METHOD PUBLIC updateCmds : BOOL
VAR_IN_OUT CONSTANT
	i_cartCtrlCmd : ST_SlaveArmCtrlCmds;
END_VAR
VAR
	i:INT;
END_VAR
m_cmdJntTrq:=i_cartCtrlCmd.m_cmdJntTrq;
m_cmdJntPos :=i_cartCtrlCmd.m_cmdJntPos;
m_cmdJntVel :=i_cartCtrlCmd.m_cmdJntVel;


// enable/disable joints
enable(i_cartCtrlCmd.m_jntEnableFlag);

// position/Velocity control
FOR i:=1 TO g_sJntNum DO 
	IF i_cartCtrlCmd.m_jntOPMode[i]=DriverOPMode_Pos THEN
		m_cmdJntTrq[i]:=0;
		m_cmdJntVel[i]:=0;
		m_cartJoints[i].updateCmd(DriverOPMode_Pos,m_cmdJntPos[i],m_cmdJntTrq[i],m_cmdJntVel[i]);
	ELSIF i_cartCtrlCmd.m_jntOPMode[i]=DriverOPMode_Vel THEN
		m_cmdJntTrq[i]:=0;
		m_cmdJntPos[i]:=0;
		m_cartJoints[i].updateCmd(DriverOPMode_Pos,m_cmdJntPos[i],m_cmdJntTrq[i],m_cmdJntVel[i]);
	ELSIF i_cartCtrlCmd.m_jntOPMode[i]=DriverOPMode_MZPos  THEN
		m_cmdJntTrq[i]:=0;
		m_cmdJntVel[i]:=0;
		//Input torque mode because the operating mode word for the contour position mode of the MingZhi driver is 1
		m_cartJoints[i].updateCmd(DriverOPMode_Trq,m_cmdJntPos[i],m_cmdJntTrq[i],m_cmdJntVel[i]);
	ELSIF i_cartCtrlCmd.m_jntOPMode[i]=DriverOPMode_cspMZ  THEN
		 m_cartJoints[i].updateCmd(DriverOPMode_cspMZ,m_cmdJntPos[i],m_cmdJntTrq[i],m_cmdJntVel[i]);
	ELSIF DriverOPMode_csvMZ = i_cartCtrlCmd.m_jntOPMode[i] THEN
		m_cartJoints[i].updateCmd(DriverOPMode_csvMZ,m_cmdJntPos[i],m_cmdJntTrq[i],m_cmdJntVel[i]);
	END_IF
END_FOR
END_METHOD

METHOD PUBLIC updateStatus : BOOL
VAR_INPUT
END_VAR
VAR
	i:INT;
END_VAR
// update joint data
FOR i:=1 TO g_sJntNum DO
	m_cartJoints[i].updateStatus();
END_FOR

//IO output   Horizontal laser IO output   Cross laser IO output
checkIO();


// get joint data
FOR i:=1 TO g_cartJntNum DO
	m_curMotorPos[i]:=m_cartJoints[i].motorPos;
	m_curLinkPos[i]:=m_cartJoints[i].linkPos;
	m_curLinkSingle[i]:=m_cartJoints[i].linkSingle;
	m_curJntPos[i]:=m_cartJoints[i].jntPos;
	m_curJntVel[i]:=m_cartJoints[i].jntVel;
	m_curJntTrq[i]:=m_cartJoints[i].jntTrq;
	m_rawJntCurrent[i]:=m_cartJoints[i].rawCurrent;
	m_filtJntCurrent[i]:=m_cartJoints[i].filtCurrent;
	m_cmdJntCurrent[i]:=m_cartJoints[i].cmdCurrent;
END_FOR
END_METHOD

END_FUNCTION_BLOCK

// ---- FBs_Robots/FB_CartJoint.TcPOU
FUNCTION_BLOCK FB_CartJoint EXTENDS FB_JointBase
VAR_INPUT
END_VAR
VAR_OUTPUT
END_VAR
VAR
	//Cart motor output IO
	m_cartMotorOutput AT %Q*	:ST_CartMotorOutput;
	
	m_cartMotorVelSongxia AT %I*  : DINT;

	m_cmdAcc:LREAL;
	
END_VAR

METHOD cmd2motorMZ : DINT
VAR_INPUT
	i_cmd:LREAL;
	i_controlCycleTime :LREAL;
END_VAR
cmd2motorMZ:=LREAL_TO_DINT(i_cmd / m_motorEnc2PosRatio);//*i_controlCycleTime
END_METHOD

METHOD PUBLIC enableMZ : BOOL
VAR_INPUT
END_VAR
IF (MZDriverStatusWord_SwitchOnDisable AND m_motorInputs.m_statusWord) = MZDriverStatusWord_SwitchOnDisable    THEN
	m_motorOutputs.m_controlWord:=DriverCtrlWord_INIT;
	enableMZ := FALSE;
ELSIF (MZDriverStatusWord_OperationEnbale AND m_motorInputs.m_statusWord) = MZDriverStatusWord_OperationEnbale THEN
	enableMZ :=  TRUE;
ELSIF (MZDriverStatusWord_SwitchOn AND m_motorInputs.m_statusWord) =  MZDriverStatusWord_SwitchOn THEN
	m_motorOutputs.m_controlWord:=DriverCtrlWord_OP;
	enableMZ :=  FALSE;
ELSIF (MZDriverStatusWord_ReadyToSwitchOn AND m_motorInputs.m_statusWord) = MZDriverStatusWord_ReadyToSwitchOn THEN
	m_motorOutputs.m_controlWord:=DriverCtrlWord_PREOP;
	enableMZ :=  FALSE;
ELSIF (MZDriverStatusWord_Fault AND m_motorInputs.m_statusWord) = MZDriverStatusWord_Fault THEN
	m_motorOutputs.m_controlWord:=DriverCtrlWord_FaultReset;
//ELSE
//	m_motorOutputs.m_controlWord:=DriverCtrlWord_INIT;
//	enable :=  FALSE;
END_IF
END_METHOD

METHOD PUBLIC init : BOOL
VAR_INPUT
	i_jntIdx :INT;
	i_controlCycleTime :LREAL;
END_VAR
m_jntIdx:=i_jntIdx;
m_cycleTime := i_controlCycleTime;

// hardware parameters
m_motorEncoderRes :=GVL_CartMotorParameters.g_incEncoderRes[i_jntIdx];
m_linkEncoderRes :=GVL_CartMotorParameters.g_absEncoderRes[i_jntIdx];
m_motorReduction :=GVL_CartMotorParameters.g_motorReduction[i_jntIdx];
m_linkEncoderReduction :=GVL_CartMotorParameters.g_absEncoderReduction[i_jntIdx];
m_trqConst :=GVL_CartMotorParameters.g_motorTrqConst[i_jntIdx];
m_maxCurrent :=GVL_CartMotorParameters.g_motorMaxCurrent[i_jntIdx];
m_motorDir :=GVL_CartMotorParameters.g_motorDir[i_jntIdx];								
m_minJntPos	:=GVL_CartMotorParameters.g_minJntPos[i_jntIdx];
m_maxJntPos	:=GVL_CartMotorParameters.g_maxJntPos[i_jntIdx];

//link encoder calibartion data
m_linkEncoderDir :=GVL_CartJointEncoderCaliData.g_asbEncoderDir[i_jntIdx];
m_minLinkEncoder :=GVL_CartJointEncoderCaliData.g_minLinkEncoder[ i_jntIdx] - m_linkEncoderDir*GVL_CartJointEncoderCaliData.g_linkEncLimitBuffer; // expand limit
m_maxLinkEncoder :=GVL_CartJointEncoderCaliData.g_maxLinkEncoder[ i_jntIdx] + m_linkEncoderDir*GVL_CartJointEncoderCaliData.g_linkEncLimitBuffer; // expand limit
m_caliLinkEncoder :=GVL_CartJointEncoderCaliData.g_caliLinkEncoder[ i_jntIdx];
m_linkEncCaliJntPos :=GVL_CartJointEncoderCaliData.g_linkEncCaliJntPos[i_jntIdx];
m_linkEncZeroCross :=GVL_CartJointEncoderCaliData.g_linkEncZeroCross[ i_jntIdx];
m_multiCycles :=GVL_CartJointEncoderCaliData.g_multipleCyclesJoint[i_jntIdx];

// convert cali link encoder if joint cross zero
IF 1=m_linkEncZeroCross THEN
	IF 1=m_linkEncoderDir AND m_caliLinkEncoder < m_minLinkEncoder THEN
		m_caliLinkEncoder := GVL_CartJointEncoderCaliData.g_caliLinkEncoder[ i_jntIdx] + m_linkEncoderRes;
	ELSIF -1=m_linkEncoderDir AND m_caliLinkEncoder < m_maxLinkEncoder THEN
		m_caliLinkEncoder := GVL_CartJointEncoderCaliData.g_caliLinkEncoder[ i_jntIdx] + m_linkEncoderRes;
	END_IF
END_IF

// macro data
m_trq2CurrentRatio:=m_motorDir * 1000.0/(m_trqConst*m_motorReduction);
m_current2TrqRatio:=m_motorDir * (m_trqConst*m_motorReduction)/1000.0;
m_linkEnc2PosRatio := 2*PI*m_linkEncoderDir/(m_linkEncoderReduction*m_linkEncoderRes);
m_motorEnc2PosRatio := 2*PI * m_motorDir/(m_motorReduction * m_motorEncoderRes);


// motor data init
m_rawJntVel :=0;
m_curJntVel:=0;
m_curJntTrq :=0;
m_rawCurrent :=0;
m_filtCurrent :=0;
m_cmdJntVel :=0.0;
m_cmdJntTrq :=0.0;
m_cmdCurrent := 0.0;

// filter init
m_jntVelLpf.init(1, GVL_CartControlParameters.g_curJntVelLpfCutoffFreq, g_cartCtrlFreq);
m_cmdTrqLpf.init(1, GVL_CartControlParameters.g_cmdJntTrqLpfCutoffFreq, g_cartCtrlFreq);
m_curTrqLpf.init(1, GVL_CartControlParameters.g_curJntTrqLpfCutoffFreq, g_cartCtrlFreq);

// driver init value
m_motorOutputs.m_controlWord:=DriverCtrlWord_INIT;
m_motorOutputs.m_opMode:=INT_TO_SINT(DriverOPMode_Pos);
m_motorOutputs.m_cmdCurrent:=0;
m_motorOutputs.m_cmdMotorEncoder:=m_motorInputs.m_motorEncoder;
END_METHOD

METHOD PUBLIC updateCmd : BOOL
VAR_INPUT
	i_opMode : E_DriverOPMode;
	i_cmdPos :LREAL;
	i_cmdTrq :LREAL;
	i_cmdVel :LREAL;
END_VAR
VAR
	i:INT;
END_VAR
m_motorOutputs.m_opMode:=INT_TO_SINT( i_opMode);

// pos mode
IF i_opMode = DriverOPMode_Pos OR i_opMode = DriverOPMode_cspMZ  THEN
	m_motorOutputs.m_cmdCurrent:=0;
	m_cmdJntPos :=i_cmdPos;
	m_cartMotorOutput.m_cmdVelMzVelMode :=0;
	m_motorOutputs.m_cmdMotorEncoder :=motorPos2Enc(m_cmdJntPos);
ELSIF i_opMode = DriverOPMode_Vel THEN
	m_cmdJntVel := i_cmdVel;
	m_cartMotorOutput.m_cmdVelMzVelMode := cmd2motorMZ(m_cmdJntVel, g_cartCtrlCycleTime);
	
ELSIF i_opMode = DriverOPMode_Trq THEN   //Here the torque mode is equal to the contour position mode of the MingZhi driver
	m_cmdJntVel := i_cmdVel;
	m_cmdAcc:=i_cmdVel*2;
	m_cmdJntPos:=i_cmdPos;
	m_cartMotorOutput.m_cmdAccMz :=cmd2motorMZ(m_cmdAcc, g_cartCtrlCycleTime);
	//m_cartMotorOutput.m_cmdVelMz := cmd2motorMZ(m_cmdJntVel, g_cartCtrlCycleTime);
	m_motorOutputs.m_cmdMotorEncoder := motorPos2Enc(m_cmdJntVel);
ELSIF i_opMode = DriverOPMode_csvMZ THEN
	m_cmdJntVel := i_cmdVel;
	m_cartMotorOutput.m_cmdVelMzVelMode := cmd2motorMZ(m_cmdJntVel, g_cartCtrlCycleTime);
	m_cartMotorOutput.m_cmdVelMax := 419430400;
END_IF
END_METHOD

METHOD PUBLIC updateStatus : BOOL
VAR_INPUT
END_VAR
// compute joint position
m_curLinkPos:= linkEnc2Pos();
m_curMotorPos:=motorEnc2Pos();
m_curLinkSingle := m_curLinkPos - 2*PI* m_linkEncCycles;

// Cart joint1-4 have no link enconder, use motor position
IF m_jntIdx <= 8 THEN
	m_curJntPos := m_curMotorPos;
ELSE
	m_curJntPos := m_curLinkPos;
END_IF

// compute joint velocity
m_curVelCalCycles := m_curVelCalCycles+1;
IF m_curVelCalCycles > m_velCalcCycles THEN
	m_rawJntVel:= (m_curJntPos-m_lastJntPos)/(m_cycleTime*m_velCalcCycles);
	m_curJntVel := m_jntVelLpf.run(m_rawJntVel);
	m_lastJntPos :=m_curJntPos;	
	m_curVelCalCycles:=1;
END_IF

IF m_jntIdx = 3 OR  m_jntIdx = 4 THEN
	m_curJntVel := m_cartMotorVelSongxia * m_motorEnc2PosRatio;
END_IF

// current and torque
m_rawCurrent := m_motorInputs.m_current;
m_filtCurrent := m_curTrqLpf.run(m_rawCurrent);
m_curJntTrq := m_filtCurrent * m_current2TrqRatio;
END_METHOD

END_FUNCTION_BLOCK

// ---- FBs_Robots/FB_JointBase.TcPOU
FUNCTION_BLOCK FB_JointBase
VAR_INPUT
END_VAR
VAR_OUTPUT
END_VAR
VAR
	// arm and joint index
	m_armIdx :INT;
	m_jntIdx :INT;
	
	// motor IO
	m_motorInputs AT%I*	:ST_MotorInputs;
	m_motorOutputs AT%Q* :ST_MotorOutputs;
	
	// cycle time
	m_cycleTime :LREAL;
	
	// calibrated link encoder data
	m_minLinkEncoder :DINT;
	m_maxLinkEncoder :DINT;
	m_caliLinkEncoder :DINT;
	m_linkEncCaliJntPos :LREAL;
	m_linkEncZeroCross :INT;
	m_initMotorEnc : DINT;
	m_multiCycles :INT;
	
	// joint position from link encoder after power on
	m_initLinkPos :LREAL;
	
	// data for link encoder multiple cycles
	m_lastLinkEncoder :DINT;
	m_linkEncCycles:INT;
	
	// device paramters
	m_motorEncoderRes :DINT;
	m_linkEncoderRes :DINT;
	m_linkEncLimitBuffer : DINT;
	m_motorReduction :LREAL;
	m_linkEncoderReduction :LREAL;
	m_trqConst :LREAL;
	m_maxCurrent :LREAL;
	m_motorDir :INT;								
	m_linkEncoderDir :INT;
	m_minJntPos: LREAL;
	m_maxJntPos: LREAL;
	
	// macro defined data for quick calculation
	m_trq2CurrentRatio:LREAL;
	m_current2TrqRatio:LREAL;
	m_linkEnc2PosRatio :LREAL;
	m_motorEnc2PosRatio :LREAL;
	
	// joint data
	m_curMotorPos :LREAL;
	m_curLinkPos :LREAL;
	m_curLinkSingle :LREAL;//[0-360]
	m_curJntPos	:LREAL;
	m_curJntVel :LREAL;
	m_rawJntVel :LREAL;
	m_curJntTrq :	LREAL;
	m_rawCurrent : LREAL;
	m_filtCurrent : LREAL;
	m_cmdJntPos :LREAL;
	m_cmdJntVel :LREAL;
	m_cmdJntTrq :LREAL;
	m_cmdCurrent : LREAL;
	m_lastJntPos :LREAL;
	
	// velocity filter
	m_jntVelLpf :FB_LowPassFilter;
	
	// command torque filter
	m_curTrqLpf : FB_LowPassFilter;
	m_cmdTrqLpf :FB_LowPassFilter;
	
	// velocity is calculated every (m_velCalcCycles) control cycles
	// TODO: insturment joint motor can not reach 4k now, so calculate their velocity with 1k frequency, need to remove later
	m_velCalcCycles :INT :=1;
	m_curVelCalCycles :INT :=1;
	
	// SDO writer
	m_opModeSDOWrite:FB_EcCoESdoWrite;
	m_MotorCurrentSDOWrite:FB_EcCoESdoWrite;
	
END_VAR

PROPERTY cmdCurrent : LREAL
GET
cmdCurrent:=m_cmdCurrent;
END_GET
END_PROPERTY

METHOD PUBLIC disable : BOOL
VAR_INPUT
END_VAR
m_motorOutputs.m_controlWord:=DriverCtrlWord_INIT;
disable:=true;
END_METHOD

METHOD PUBLIC enable : BOOL
VAR_INPUT
END_VAR
IF DriverStatusWord_INIT = m_motorInputs.m_statusWord THEN
	m_motorOutputs.m_controlWord:=DriverCtrlWord_PREOP;
	enable := FALSE;
ELSIF DriverStatusWord_PREOP = m_motorInputs.m_statusWord THEN
	m_motorOutputs.m_controlWord:=DriverCtrlWord_OP;
	enable :=  FALSE;
ELSIF DriverStatusWord_OP = m_motorInputs.m_statusWord THEN
	enable :=  TRUE;
//ELSE
//	m_motorOutputs.m_controlWord:=DriverCtrlWord_INIT;
//	enable :=  FALSE;
END_IF
END_METHOD

PROPERTY filtCurrent : LREAL
GET
filtCurrent:=m_filtCurrent;
END_GET
END_PROPERTY

METHOD PUBLIC initJntPos : BOOL
VAR_INPUT
END_VAR
m_lastLinkEncoder :=m_motorInputs.m_linkEncoder;
m_linkEncCycles:=0;
m_curLinkPos :=linkEnc2Pos();
m_initLinkPos:=m_curLinkPos;
m_initMotorEnc :=m_motorInputs.m_motorEncoder;
m_curMotorPos:=motorEnc2Pos();
m_curJntPos := m_curMotorPos;
m_cmdJntPos :=m_curJntPos;	
m_lastJntPos :=m_curJntPos;
END_METHOD

PROPERTY initLinkPos : lreal
GET
initLinkPos:=m_initLinkPos;
END_GET
SET
m_initLinkPos:=initLinkPos;
END_SET
END_PROPERTY

METHOD PUBLIC isEnabled : BOOL
VAR_INPUT
END_VAR
isEnabled :=(DriverStatusWord_OP = m_motorInputs.m_statusWord);
END_METHOD

PROPERTY jntPos : LREAL
GET
jntPos := m_curJntPos;
END_GET
END_PROPERTY

PROPERTY jntTrq : LREAL
GET
jntTrq:=m_curJntTrq;
END_GET
END_PROPERTY

PROPERTY jntVel : LREAL
GET
jntVel := m_curJntVel;
END_GET
END_PROPERTY

METHOD PROTECTED linkEnc2Pos : LREAL
VAR_INPUT
END_VAR
VAR
	incLinkPos :LREAL;
	newLinkEnc :DINT;
END_VAR
// cycle check
IF 1=m_multiCycles THEN
	IF (m_motorInputs.m_linkEncoder - m_lastLinkEncoder)*m_linkEncoderDir < -m_linkEncoderRes/2 THEN
		m_linkEncCycles :=m_linkEncCycles+1;
	ELSIF (m_motorInputs.m_linkEncoder - m_lastLinkEncoder)*m_linkEncoderDir > m_linkEncoderRes/2 THEN
		m_linkEncCycles :=m_linkEncCycles-1;
	END_IF
END_IF
m_lastLinkEncoder:=m_motorInputs.m_linkEncoder;

// convert link encoder if joint cross zero
newLinkEnc := m_motorInputs.m_linkEncoder;
IF 1=m_linkEncZeroCross AND 0 = m_multiCycles THEN
	IF 1=m_linkEncoderDir AND m_motorInputs.m_linkEncoder < m_minLinkEncoder THEN
		newLinkEnc := m_motorInputs.m_linkEncoder + m_linkEncoderRes;
	ELSIF -1=m_linkEncoderDir AND m_motorInputs.m_linkEncoder < m_maxLinkEncoder THEN
		newLinkEnc := m_motorInputs.m_linkEncoder + m_linkEncoderRes;
	END_IF
END_IF

// motion from calibrated points
incLinkPos := (newLinkEnc-m_caliLinkEncoder)*m_linkEnc2PosRatio;

// absolute joint position
linkEnc2Pos := incLinkPos + m_linkEncCaliJntPos + 2*PI* m_linkEncCycles;
END_METHOD

PROPERTY PUBLIC linkPos : LREAL
GET
linkPos:=m_curLinkPos;
END_GET
END_PROPERTY

PROPERTY linkSingle : LREAL
GET
linkSingle :=m_curLinkSingle;
END_GET
END_PROPERTY

METHOD PROTECTED motorEnc2Pos : LREAL
VAR_INPUT
END_VAR
motorEnc2Pos:= (m_motorInputs.m_motorEncoder-m_initMotorEnc)* m_motorEnc2PosRatio +m_initLinkPos;
END_METHOD

PROPERTY PUBLIC motorPos : LREAL
GET
motorPos := m_curMotorPos;
END_GET
END_PROPERTY

METHOD PROTECTED motorPos2Enc : DINT
VAR_INPUT
	i_jntPos :LREAL;
END_VAR

VAR
END_VAR

motorPos2Enc := LREAL_TO_DINT((i_jntPos-m_initLinkPos)/m_motorEnc2PosRatio + m_initMotorEnc);
END_METHOD

PROPERTY rawCurrent : LREAL
GET
rawCurrent := m_rawCurrent;
END_GET
END_PROPERTY

METHOD PROTECTED singleCyclePos : LREal
VAR_INPUT
END_VAR
VAR
	cycles :lreal;
END_VAR
cycles := ABS(FLOOR( m_curJntPos/g_2pi));
IF m_curJntPos<0 THEN
	singleCyclePos := m_curJntPos+cycles*g_2pi;
ELSE
	singleCyclePos := m_curJntPos-cycles*g_2pi;
END_IF
END_METHOD

METHOD PUBLIC updateCmds : BOOL
VAR_INPUT
	i_opMode : E_DriverOPMode;
	i_cmdPos :LREAL;
	i_cmdTrq :LREAL;
END_VAR
VAR
	filtCmdTrq :LREAL;
END_VAR
m_motorOutputs.m_opMode:=INT_TO_SINT( i_opMode);
// pos mode
IF i_opMode = DriverOPMode_Pos THEN
	m_motorOutputs.m_cmdCurrent:=0;
	m_cmdTrqLpf.reset();	
//	i_cmdPos:=LIMIT(m_minJntPos, i_cmdPos, m_maxJntPos); // May cause position jump, Do this in safety check. 
	m_cmdJntPos :=i_cmdPos;
	m_motorOutputs.m_cmdMotorEncoder :=motorPos2Enc(m_cmdJntPos);
ELSIF i_opMode = DriverOPMode_Trq THEN
	filtCmdTrq:=m_cmdTrqLpf.run(i_cmdTrq);
	m_motorOutputs.m_cmdCurrent:=LREAL_TO_DINT(LIMIT(-m_maxCurrent, filtCmdTrq*m_trq2CurrentRatio,m_maxCurrent));
	m_motorOutputs.m_cmdMotorEncoder :=m_motorInputs.m_motorEncoder; 
END_IF
m_cmdCurrent:=m_motorOutputs.m_cmdCurrent;
END_METHOD

METHOD PUBLIC updateStatus : BOOL
VAR_INPUT
END_VAR
// compute joint position
m_curLinkPos:= linkEnc2Pos();
m_curMotorPos:=motorEnc2Pos();
m_curJntPos := m_curMotorPos;
m_curLinkSingle := singleCyclePos();

// compute joint velocity
m_curVelCalCycles := m_curVelCalCycles+1;
IF m_curVelCalCycles > m_velCalcCycles THEN
	m_rawJntVel:= (m_curJntPos-m_lastJntPos)/(m_cycleTime*m_velCalcCycles);
	m_curJntVel := m_jntVelLpf.run(m_rawJntVel);
	m_lastJntPos :=m_curJntPos;	
	m_curVelCalCycles:=1;
END_IF


// current and torque
m_rawCurrent := m_motorInputs.m_current;
m_filtCurrent := m_curTrqLpf.run(m_rawCurrent);
m_curJntTrq := m_filtCurrent * m_current2TrqRatio;
END_METHOD

END_FUNCTION_BLOCK

// ---- FBs_CartControlles/FB_CartCtrlAdjust.TcPOU
FUNCTION_BLOCK FB_CartCtrlAdjust EXTENDS FB_CartCtrlBase
VAR_INPUT
END_VAR
VAR_OUTPUT
END_VAR
VAR

	m_joystickSignal: Vec8d;	
	m_fiducialValue:INT:= 512;
	m_joystickRange:INT:=430;
	m_joystickDir: Vec8i:=[1,1,1,1,-1,-1,1,1];
	m_joystickVelInc: Vec8d;
	m_actJntPos: Vec8d;
	m_tarPosInc: Vec8d;
	m_lastPosInc: Vec8d;
	m_tarCartPos: Vec8d;
	m_trajJntPos : Vec8d;
	m_tarJntPos : Vec8d;
	m_initActJntPos: Vec8d;
	m_initActCartPos: Vec8d;
	m_veiwAngle : LREAL;
	m_jntPosReachLimit : Vec8b;
	m_maxJntPos : vec8d;

	m_carJntSoftwareLimit :ARRAY [5..8] OF LREAL := [0.005, 2*g_deg2Rad, 0.005, 2*g_deg2Rad];
	
	// time threshold to 5-8joint after it's enabled
	m_cartAdjustStartWaitTime :LREAL := 0.3;
	
	//adjust start  time 
	m_adjustStartTime :LREAL;
	
	// filter cut-off frequency for cart drive force 
	m_cmdJoystickLpfCutoffFreq : LREAL :=8;
	m_cartCtrlFreq :LREAL:=8000;
	
	m_Vel : LREAL;
	m_velDir : INT;
	m_jntOTG :ARRAY[1..8] OF FB_secOrdTrajFilter;
END_VAR

// override this function in each exact controller
METHOD PROTECTED calcCmdJntPos : BOOL
VAR_IN_OUT CONSTANT
	// slave cart joint data
	i_slaveCart :FB_SlaveCart;
END_VAR

VAR
	i:INT;
END_VAR
//In this method, 5 represents the pillar postion , 6 represents the beam rotation angle ,7 represents the beam stretch position ,8 represents the overhang angle
m_adjustStartTime :=LIMIT(0, m_adjustStartTime + g_cartCtrlCycleTime, 1);
m_actJntPos := i_slaveCart.curJntPos;
m_actJntPos[7] := i_slaveCart.curJntPos[7] + GVL_CartControlParameters.g_curBeamStretchJntInitPos;
m_veiwAngle := m_actJntPos[6] + m_actJntPos[8];

IF m_adjustStartTime > m_cartAdjustStartWaitTime THEN
	FOR i:= 1 TO 4 BY 1 DO
		m_joystickSignal[i] := i_slaveCart.m_joystickSignal[i] - m_fiducialValue;
		m_joystickVelInc[i+4] := m_joystickSignal[i]/m_joystickRange*m_joystickDir[i+4]*GVL_CartControlParameters.g_maxCartVel[i];
		m_tarPosInc[i+4] := m_tarPosInc[i+4] + m_joystickVelInc[i+4] * g_cartCtrlCycleTime;
	END_FOR
	
	m_tarCartPos[5] := m_initActJntPos[5] + m_tarPosInc[5];
	IF i_slaveCart.m_ctrlEnable.m_cameraJoystickEnable THEN
		m_tarCartPos[6] := m_initActCartPos[6] + m_tarPosInc[6]*COS(m_veiwAngle)+m_tarPosInc[7]*SIN(m_veiwAngle);
		m_tarCartPos[7] := m_initActCartPos[7] - m_tarPosInc[6]*SIN(m_veiwAngle)+m_tarPosInc[7]*COS(m_veiwAngle);
	ELSE
		m_tarCartPos[6] := m_initActCartPos[6] + m_tarPosInc[6];
		m_tarCartPos[7] := m_initActCartPos[7] + m_tarPosInc[7];
	END_IF
	m_tarCartPos[8] := m_initActJntPos[8] + m_tarPosInc[8];
	
	IF i_slaveCart.m_ctrlEnable.m_heightLimitAdjustEnable THEN
		m_trajJntPos[5] := m_tarCartPos[5];
	ELSE
		m_trajJntPos[5] := LIMIT(GVL_CartMotorParameters.g_minJntPos[5], m_tarCartPos[5], MAX(m_actJntPos[5],i_slaveCart.m_cartDataFromUI.m_standColumnHightLimit));
	END_IF
	m_trajJntPos[6] := atan2( m_tarCartPos[6], m_tarCartPos[7]);
	m_trajJntPos[7] := m_tarCartPos[7]/COS(m_trajJntPos[6]) - GVL_CartControlParameters.g_curBeamStretchJntInitPos;
	m_trajJntPos[8] := m_tarCartPos[8] -  (m_trajJntPos[6] - m_initActJntPos[6]);
	m_jntPosReachLimit := calcCmdReachLimit();
	m_jntEnableFlag := faultDetect(i_slaveCart.curJntPos);
	FOR i := 5 TO 8 DO 
		m_tarJntPos[i] := LIMIT(GVL_CartMotorParameters.g_minJntPos[i] + m_carJntSoftwareLimit[i], m_trajJntPos[i], GVL_CartMotorParameters.g_maxJntPos[i] - m_carJntSoftwareLimit[i]) ;
		m_jntOTG[i].run(i_targetPos:= m_trajJntPos[i], i_targetVel:= 0.0, o_cmdAcc=> , o_cmdVel=> , o_cmdPos=>m_cmdJntPos[i] );
	END_FOR
END_IF
END_METHOD

METHOD calcCmdReachLimit : vec8b
VAR_INPUT
END_VAR

VAR
	i : INT;
END_VAR

FOR i := 5 TO g_cartJntNum DO
	IF (GVL_CartMotorParameters.g_minJntPos[i] + m_carJntSoftwareLimit[i]) >= m_trajJntPos[i] THEN
		IF (m_tarPosInc[i] - m_lastPosInc[i]) <0 THEN
			m_tarPosInc[i] := m_lastPosInc[i];
		END_IF
		calcCmdReachLimit[i] := TRUE;
	
	ELSIF m_trajJntPos[i]>=(m_maxJntPos[i] - m_carJntSoftwareLimit[i]) THEN
		IF (m_tarPosInc[i] - m_lastPosInc[i]) >0 THEN
			m_tarPosInc[i] := m_lastPosInc[i];
		END_IF
		calcCmdReachLimit[i] := TRUE;
	END_IF
	m_lastPosInc[i] := m_tarPosInc[i];
END_FOR
END_METHOD

METHOD faultDetect : vec8i
VAR_INPUT
	curJntPos : vec8d;
END_VAR
faultDetect[5] := BOOL_TO_INT( NOT SafetyCheck.m_safetyCheckData.m_cartStandColumnErr);
faultDetect[6] := BOOL_TO_INT( NOT SafetyCheck.m_safetyCheckData.m_cartAdjustErr);
faultDetect[7] := BOOL_TO_INT( NOT SafetyCheck.m_safetyCheckData.m_cartAdjustErr);
faultDetect[8] := BOOL_TO_INT( NOT SafetyCheck.m_safetyCheckData.m_cartAdjustErr);

IF SafetyCheck.m_safetyCheckData.m_cartStandColumnErr THEN
	m_trajJntPos[5] :=curJntPos[5];
END_IF
IF SafetyCheck.m_safetyCheckData.m_cartAdjustErr THEN
	m_trajJntPos[6] :=curJntPos[6];
	m_trajJntPos[7] :=curJntPos[7];
	m_trajJntPos[8] :=curJntPos[8];
END_IF
END_METHOD

// override this function in each exact controller
// NOTICE: set joint control mode here, and do some initialization if needed
METHOD PUBLIC init : BOOL
VAR_IN_OUT CONSTANT
	i_slaveCart	:FB_SlaveCart;
END_VAR
VAR_IN_OUT 
	r_cartCtrlCmd :ST_SlaveArmCtrlCmds;
END_VAR
VAR
	i:INT;
END_VAR
// check if to hold the command joint position unchanged
//m_holdLastCmds := checkToHoldLastCmds(i_slaveCart);
m_holdLastCmds := checkToHoldLastCmds(i_slaveCart);
SUPER^.init(i_slaveCart,r_cartCtrlCmd);

m_jntEnableFlag[5] := BOOL_TO_INT( NOT SafetyCheck.m_safetyCheckData.m_cartStandColumnErr);
m_jntEnableFlag[6] := BOOL_TO_INT( NOT SafetyCheck.m_safetyCheckData.m_cartAdjustErr);
m_jntEnableFlag[7] := BOOL_TO_INT( NOT SafetyCheck.m_safetyCheckData.m_cartAdjustErr);
m_jntEnableFlag[8] := BOOL_TO_INT( NOT SafetyCheck.m_safetyCheckData.m_cartAdjustErr);

m_jntOPMode[5]:= DriverOPMode_cspMZ;
m_jntOPMode[6]:= DriverOPMode_Pos;
m_jntOPMode[7]:= DriverOPMode_Pos;
m_jntOPMode[8]:= DriverOPMode_Pos;

m_joystickSignal := g_zeroVec8d;
m_tarPosInc := g_zeroVec8d;
m_trajJntPos := g_zeroVec8d;
m_lastPosInc := g_zeroVec8d;
m_jntPosReachLimit := g_zeroVec8b;

m_maxJntPos := GVL_CartMotorParameters.g_maxJntPos;
m_maxJntPos[5] := i_slaveCart.m_cartDataFromUI.m_standColumnHightLimit;

m_initActJntPos:=m_cmdJntPos;//i_slaveCart.curJntPos;
m_initActCartPos[6] := (m_initActJntPos[7] + GVL_CartControlParameters.g_curBeamStretchJntInitPos) * SIN(m_initActJntPos[6]);
m_initActCartPos[7] := (m_initActJntPos[7] + GVL_CartControlParameters.g_curBeamStretchJntInitPos) * COS(m_initActJntPos[6]);

FOR i := 1 TO 4 BY 1 DO
	m_jntOTG[i+4].init(i_curCmdPos:= m_cmdJntPos[i+4], i_curCmdVel:= 0, i_maxV:=GVL_CartControlParameters.g_maxJntVel[i+4] , i_maxA:=GVL_CartControlParameters.g_maxJntAcc[i+4] , i_Ts:=g_cartCtrlCycleTime );
END_FOR

m_adjustStartTime := 0;
// update commands to arm
copyCmds(r_cartCtrlCmd);
END_METHOD

PROPERTY jntPosReachLimit : vec8b
GET
jntPosReachLimit := m_jntPosReachLimit;
END_GET
END_PROPERTY

END_FUNCTION_BLOCK

// ---- FBs_CartControlles/FB_CartCtrlSlowDown.TcPOU
FUNCTION_BLOCK FB_CartCtrlSlowDown EXTENDS FB_CartCtrlBase
VAR_INPUT
END_VAR
VAR_OUTPUT
END_VAR
VAR

	m_tarPosInc: Vec8d;
	m_trajVel : Vec8d;
	m_initVel : Vec8d;
	m_initPos : Vec8d;
	m_initDec : Vec8d;
	
	//slow down and stop time
	m_incSlowStopTime :LREAL;
	m_slowStopTime :LREAL :=0.5;
	
	// filter cut-off frequency for cart drive force 
	m_cmdJoystickLpfCutoffFreq : LREAL :=8;
	m_cartCtrlFreq :LREAL:=8000;
END_VAR

// override this function in each exact controller
METHOD PROTECTED calcCmdJntPos : BOOL
VAR_IN_OUT CONSTANT
	// slave cart joint data
	i_slaveCart :FB_SlaveCart;
END_VAR

VAR
	i:INT;
END_VAR
//In this method, 5 represents the pillar postion , 6 represents the beam rotation angle ,7 represents the beam stretch position ,8 represents the overhang angle
m_incSlowStopTime :=LIMIT(0, m_incSlowStopTime + g_cartCtrlCycleTime, 1);

FOR i := 5 TO 8 BY 1 DO
	m_trajVel[i] := m_initVel[i] - m_initDec[i] * m_incSlowStopTime;
	IF sign(m_trajVel[i]) <> sign(m_initVel[i]) THEN
		m_trajVel[i]:=0;
	END_IF
	m_tarPosInc[i] := m_tarPosInc[i] + m_trajVel[i] * g_cartCtrlCycleTime;
	m_cmdJntPos[i] := m_initPos[i] + m_tarPosInc[i];
END_FOR

IF m_incSlowStopTime >= m_slowStopTime THEN//m_slowStopTime THEN
	m_isFinished := TRUE;
END_IF
END_METHOD

// override this function in each exact controller
METHOD PROTECTED calcCmdJntVel : BOOL
VAR_IN_OUT CONSTANT
	// slave cart joint data
	i_slaveCart :FB_SlaveCart;
END_VAR

VAR
	i:INT;
END_VAR
//In this method, 5 represents the pillar postion , 6 represents the beam rotation angle ,7 represents the beam stretch position ,8 represents the overhang angle
m_incSlowStopTime :=LIMIT(0, m_incSlowStopTime + g_cartCtrlCycleTime, 1);

FOR i := 3 TO 4 BY 1 DO
	m_trajVel[i] := m_initVel[i] - m_initDec[i] * m_incSlowStopTime;
	IF sign(m_trajVel[i]) <> sign(m_initVel[i]) THEN
		m_trajVel[i]:=0;
	END_IF
	m_cmdJntVel[i] := LIMIT(-GVL_CartControlParameters.g_maxJntVel[i], m_trajVel[i]  , GVL_CartControlParameters.g_maxJntVel[i]);
END_FOR

IF m_incSlowStopTime >= m_slowStopTime THEN//m_slowStopTime THEN
	m_isFinished := TRUE;
END_IF
END_METHOD

// override this function in each exact controller
// NOTICE: set joint control mode here, and do some initialization if needed
METHOD PUBLIC init : BOOL
VAR_IN_OUT CONSTANT
	i_slaveCart	:FB_SlaveCart;
END_VAR
VAR_IN_OUT 
	r_cartCtrlCmd :ST_SlaveArmCtrlCmds;
END_VAR
m_cmdJntPos:=r_cartCtrlCmd.m_cmdJntPos;
m_initPos := m_cmdJntPos;

m_jntEnableFlag :=r_cartCtrlCmd.m_jntEnableFlag;

m_jntOPMode[3]:= DriverOPMode_csvMZ;
m_jntOPMode[4]:= DriverOPMode_csvMZ;
m_jntOPMode[5]:= DriverOPMode_cspMZ;
m_jntOPMode[6]:= DriverOPMode_Pos;
m_jntOPMode[7]:= DriverOPMode_Pos;
m_jntOPMode[8]:= DriverOPMode_Pos;

m_trajVel[3] := 0;
m_trajVel[4] := 0;
m_trajVel[5] := 0;
m_trajVel[6] := 0;
m_trajVel[7] := 0;
m_trajVel[8] := 0;

m_tarPosInc[3] := 0;
m_tarPosInc[4] := 0;
m_tarPosInc[5] := 0;
m_tarPosInc[6] := 0;
m_tarPosInc[7] := 0;
m_tarPosInc[8] := 0;


m_incSlowStopTime := 0;

m_initVel[3] := LIMIT(-GVL_CartControlParameters.g_maxJntVel[3], i_slaveCart.curJntVel[3], GVL_CartControlParameters.g_maxJntVel[3]);
m_initVel[4] := LIMIT(-GVL_CartControlParameters.g_maxJntVel[4], i_slaveCart.curJntVel[4], GVL_CartControlParameters.g_maxJntVel[4]);
m_initVel[5] := LIMIT(-GVL_CartControlParameters.g_maxJntVel[5], i_slaveCart.curJntVel[5], GVL_CartControlParameters.g_maxJntVel[5]);
m_initVel[6] := LIMIT(-GVL_CartControlParameters.g_maxJntVel[6], i_slaveCart.curJntVel[6], GVL_CartControlParameters.g_maxJntVel[6]);
m_initVel[7] := LIMIT(-GVL_CartControlParameters.g_maxJntVel[7], i_slaveCart.curJntVel[7], GVL_CartControlParameters.g_maxJntVel[7]);
m_initVel[8] := LIMIT(-GVL_CartControlParameters.g_maxJntVel[8], i_slaveCart.curJntVel[8], GVL_CartControlParameters.g_maxJntVel[8]);

m_initDec[3] := m_initVel[3]*2;
m_initDec[4] := m_initVel[4]*2;
m_initDec[5] := sign(m_initVel[5])*GVL_CartControlParameters.g_maxJntVel[5]*2;
m_initDec[6] := sign(m_initVel[6])*GVL_CartControlParameters.g_maxJntVel[6]*2;
m_initDec[7] := sign(m_initVel[7])*GVL_CartControlParameters.g_maxJntVel[7]*2;
m_initDec[8] := sign(m_initVel[8])*GVL_CartControlParameters.g_maxJntVel[8]*2;

m_slowStopTime := 0.5;
// update commands to arm
copyCmds(r_cartCtrlCmd);
END_METHOD

END_FUNCTION_BLOCK

// ---- FBs_CartControlles/FB_CartSupporLeg.TcPOU
FUNCTION_BLOCK FB_CartSupporLeg EXTENDS FB_CartCtrlBase
VAR_INPUT
END_VAR
VAR_OUTPUT
END_VAR
VAR

	m_actJntPos: Vec8d;
	m_tarJntPos: Vec8d;
	m_initJntPos : Vec8d;
	m_tarJntInc : Vec8d;
	m_maxJntCurrent : ARRAY [1..2] OF LREAL := [800,800];
	m_pinDeployed : ARRAY [1..2] OF BOOL; 
	
	// time threshold to 5-8joint after it's enabled
	m_cartAdjustStartWaitTime :LREAL := 0.2;
	
	//adjust start  time 
	m_adjustStartTime :LREAL;

	m_jntOTG :ARRAY [1..2] OF FB_secOrdTrajFilter;
END_VAR

// override this function in each exact controller
METHOD PROTECTED calcCmdJntPos : BOOL
VAR_IN_OUT CONSTANT
	// slave cart joint data
	i_slaveCart :FB_SlaveCart;
END_VAR

VAR
	i:INT;
END_VAR
//In this method, 8 represents the overhang angle
m_adjustStartTime :=LIMIT(0, m_adjustStartTime + g_cartCtrlCycleTime, 2);
m_actJntPos := i_slaveCart.curJntPos;
IF m_adjustStartTime > m_cartAdjustStartWaitTime THEN
	FOR i:=1 TO 2 DO
		IF ABS(i_slaveCart.curJntCurrent[i]) > m_maxJntCurrent[i] AND ABS(i_slaveCart.curJntVel[i]) < 0.002 and m_adjustStartTime >= 2  THEN
			m_pinDeployed[i] := TRUE;
			m_tarJntPos[i] := m_actJntPos[i];
		END_IF
		
		IF FALSE = m_pinDeployed[i] THEN
			m_tarJntPos[i] := m_actJntPos[i] - GVL_CartControlParameters.g_maxJntVel[i] * 2 * g_cartCtrlCycleTime;
		END_IF
		m_jntOTG[i].run(i_targetPos:= m_tarJntPos[i], i_targetVel:= 0.0, o_cmdAcc=> , o_cmdVel=> , o_cmdPos=>m_cmdJntPos[i] );
	END_FOR
	
	IF m_pinDeployed[1] AND m_pinDeployed[2] THEN
		m_isFinished := TRUE;
	END_IF

END_IF
END_METHOD

// override this function in each exact controller
// NOTICE: set joint control mode here, and do some initialization if needed
METHOD PUBLIC init : BOOL
VAR_IN_OUT CONSTANT
	i_slaveCart	:FB_SlaveCart;
END_VAR
VAR_IN_OUT 
	r_cartCtrlCmd :ST_SlaveArmCtrlCmds;
END_VAR
VAR
	i:INT;
END_VAR
//m_holdLastCmds := checkToHoldLastCmds(i_slaveCart);
m_holdLastCmds := checkToHoldLastCmds(i_slaveCart);

SUPER^.init(i_slaveCart,r_cartCtrlCmd);

m_jntEnableFlag[1] :=1;
m_jntEnableFlag[2] :=1;

m_jntOPMode[1]:= DriverOPMode_Pos;
m_jntOPMode[2]:= DriverOPMode_Pos;

m_pinDeployed[1] := FALSE;
m_pinDeployed[2] := FALSE;

m_jntOTG[1].init(i_curCmdPos:= m_cmdJntPos[1], i_curCmdVel:= 0, i_maxV:=GVL_CartControlParameters.g_maxJntVel[1] , i_maxA:=GVL_CartControlParameters.g_maxJntAcc[1] , i_Ts:=g_cartCtrlCycleTime );
m_jntOTG[2].init(i_curCmdPos:= m_cmdJntPos[2], i_curCmdVel:= 0, i_maxV:=GVL_CartControlParameters.g_maxJntVel[2] , i_maxA:=GVL_CartControlParameters.g_maxJntAcc[2] , i_Ts:=g_cartCtrlCycleTime );

m_adjustStartTime := 0;
// update commands to arm
copyCmds(r_cartCtrlCmd);
END_METHOD

END_FUNCTION_BLOCK

// ---- FBs_Auxiliary/FB_setupJnt5AdjustDetect.TcPOU
FUNCTION_BLOCK FB_setupJnt5AdjustDetect
VAR_INPUT
END_VAR
VAR_OUTPUT
END_VAR
VAR
	m_pAutoAdjustOnCounts :INT :=0;
	m_nAutoAdjustOnCounts :INT :=0;
	m_adjustOnCountThres :INT :=50;
END_VAR

METHOD run : INT
VAR_INPUT
	IOValue :UDINT;
END_VAR

VAR_OUTPUT
	
END_VAR
// joint3 positive auto adjust is 3th bit
IF 2=(IOValue AND 10#2) THEN
	m_pAutoAdjustOnCounts :=MIN(m_pAutoAdjustOnCounts +1,m_adjustOnCountThres);
ELSE
	m_pAutoAdjustOnCounts :=0;
END_IF

// joint3 negative auto adjust is 2th bit
IF 1=(IOValue AND 10#1) THEN
	m_nAutoAdjustOnCounts :=MIN(m_nAutoAdjustOnCounts +1,m_adjustOnCountThres);
ELSE
	m_nAutoAdjustOnCounts :=0;
END_IF

IF m_pAutoAdjustOnCounts >= m_adjustOnCountThres THEN
	run :=1;
ELSIF m_nAutoAdjustOnCounts >= m_adjustOnCountThres THEN
	run := -1;
ELSE 
	run :=0;
END_IF
END_METHOD

END_FUNCTION_BLOCK

// ---- FBs_Auxiliary/FB_PanelDetect.TcPOU
FUNCTION_BLOCK FB_PanelDetect
VAR_INPUT
END_VAR
VAR_OUTPUT
END_VAR
VAR
	m_panelOnCounts :INT :=0;
	m_panelOnCountThres :INT :=50;
END_VAR

// check if panel is on
METHOD run : BOOL
VAR_INPUT
	IOValue :UDINT;
END_VAR
//Panel single  At installation--2#0000   not installation --2#0101
IF (IOValue AND 16#06) = 0 THEN
	m_panelOnCounts := MIN( m_panelOnCounts +1,m_panelOnCountThres);
ELSIF (IOValue AND 16#06) = 6  THEN
	m_panelOnCounts :=0;
END_IF
run := m_panelOnCounts >= m_panelOnCountThres;
END_METHOD

END_FUNCTION_BLOCK

// ---- FBs_Auxiliary/FB_InstrumentDetect.TcPOU
FUNCTION_BLOCK FB_InstrumentDetect
VAR_INPUT
END_VAR
VAR_OUTPUT
END_VAR
VAR
	m_instruOnCounts :INT :=0;
	m_InstruOnCountThres :INT :=50;
END_VAR

// check if instrument is on
METHOD run : BOOL
VAR_INPUT
	IOValue :UDINT;
END_VAR
//Instrument single   At installation--2#0*0*   not installation --2#1*1*  And Hall single --2#100 0000
IF (IOValue AND 10#09) = 0  THEN
	m_instruOnCounts := MIN( m_instruOnCounts +1,m_InstruOnCountThres);
ELSIF (IOValue AND 10#09) = 9  THEN
	m_instruOnCounts :=0;
END_IF
run := m_instruOnCounts >= m_InstruOnCountThres;
END_METHOD

END_FUNCTION_BLOCK

// ---- FBs_RobotDynamics/FB_SetupGravity.TcPOU
FUNCTION_BLOCK FB_SetupGravity
VAR_INPUT
END_VAR
VAR
	m_armIdx :INT ;

	// current arm parameters
	m_armParams :ARRAY[1..7] OF LREAL;

	// gravity regression matrix
	regMat:ARRAY[1..7] OF LREAL;
	
	m_graivty :LREAL;
END_VAR

METHOD getRegMat : BOOL
VAR_INPUT
	// joint position of setup joint, joint6-8
	setupAng :LREAL;
	q1: LREAL;
	q2: LREAL;
	q3: LREAL;
END_VAR

VAR
	s0,c0,s1,c1,s2, c2,d3 :LREAL;
END_VAR

VAR_OUTPUT
	o_regMat:ARRAY[1..7] OF LREAL;
END_VAR
s0:= SIN(setUpAng);
c0:= COS(setUpAng);
s1:=SIN(q1);
c1:=COS(q1);
s2:=SIN(q2);
c2:=COS(q2);
d3:=q3;

// setup joint
o_regMat[1] :=c0;
o_regMat[2] := s0;
o_regMat[3] :=-(c2*s0*d3+c0*c1*s2*d3);
o_regMat[4] :=  -c0*c1;
o_regMat[5] :=  -c0*s1;
o_regMat[6] := - (c0*c1*s2+c2*s0);
o_regMat[7] :=  s0*s2- c0*c1*c2  ;
END_METHOD

METHOD init : BOOL
VAR_INPUT
	i_armIdx :INT;
END_VAR
m_armIdx :=i_armIdx;
END_METHOD

METHOD run : BOOL
VAR_IN_OUT CONSTANT
	// setup joint angle
	i_setupJntPos :Vec5d;
	
	// slave joint angle
	i_slaveJntPos :Vec8d;
	
	// instrument
	i_instruStatus :ST_InstruStatus;
END_VAR
VAR_OUTPUT
	// setup joint3 gravity
	o_jnt3Gravity :LREAL;
	
	// setup joint5 gravity
	o_jnt5Gravity :LREAL;
END_VAR
VAR
	setupPos, q1, q2, q3 :LREAL;
	i,j:INT;
	
	gravityTrq :Vec4d;

END_VAR
setupPos:=LIMIT(GVL_SetupMotorParameters.g_minJntPos[m_armIdx,5], i_setupJntPos[5], GVL_SetupMotorParameters.g_maxJntPos[m_armIdx,5]);
q1 :=LIMIT (GVL_SlaveMotorParameters.g_minJntPos[1], i_slaveJntPos[1], GVL_SlaveMotorParameters.g_maxJntPos[1]);
q2 := LIMIT (GVL_SlaveMotorParameters.g_minJntPos[2], i_slaveJntPos[2], GVL_SlaveMotorParameters.g_maxJntPos[2]);
q3 := LIMIT (GVL_SlaveMotorParameters.g_minJntPos[3], i_slaveJntPos[3], GVL_SlaveMotorParameters.g_maxJntPos[3]);

// get regression matrx
getRegMat(setupPos, q1, q2, q3, o_regMat=>regMat);

// determine current arm parameters
m_armParams[1] := GVL_SetupArmDynamics.g_setupJnt5GravityParam[m_armIdx,1];
m_armParams[2] := GVL_SetupArmDynamics.g_setupJnt5GravityParam[m_armIdx,2];
IF FALSE = i_instruStatus.m_ready THEN
	// arm only
	FOR i:=1 TO 5 DO
		m_armParams[i+2]:= GVL_SlaveArmDynamics.g_gravityParam[m_armIdx,i];
	END_FOR

// endoscope
ELSIF InstruType_endoscope = i_instruStatus.m_type THEN 
	FOR i:=1 TO 5 DO
		m_armParams[i+2]:=GVL_SlaveArmDynamics.g_gravityParam[m_armIdx,i]+GVL_SlaveArmDynamics.g_gravityEndoscope[i];
	END_FOR

// instrument
ELSE
	FOR i:=1 TO 5 DO
		m_armParams[i+2]:=GVL_SlaveArmDynamics.g_gravityParam[m_armIdx,i]+GVL_SlaveArmDynamics.g_gravityInstrument[i];
	END_FOR
// TODO:Trocar
END_IF

// calculate gravity torque
o_jnt5Gravity:=0;
FOR j:=1 TO 7 DO
	o_jnt5Gravity:=o_jnt5Gravity+regMat[j]*m_armParams[j];
END_FOR
m_graivty := o_jnt5Gravity;

o_jnt3Gravity:= setupJnt3Gravity(i_setupJntPos[3]);
END_METHOD

METHOD setupJnt3Gravity : LREAL
VAR_INPUT
	i_jnt3Pos :LREAL;
END_VAR
VAR
	q:LREAL;
END_VAR
q := LIMIT(GVL_SetupArmDynamics.g_setupJnt3GravityPosRange[m_armIdx,1], i_jnt3Pos, GVL_SetupArmDynamics.g_setupJnt3GravityPosRange[m_armIdx,2]);
setupJnt3Gravity:=GVL_SetupArmDynamics.g_setupJnt3GravityParams[m_armIdx,1]*EXPT(q,3)+GVL_SetupArmDynamics.g_setupJnt3GravityParams[m_armIdx,2]*EXPT(q,2)+
				GVL_SetupArmDynamics.g_setupJnt3GravityParams[m_armIdx,3]*q+GVL_SetupArmDynamics.g_setupJnt3GravityParams[m_armIdx,4];
				
setupJnt3Gravity:=-GVL_SetupMotorParameters.g_motorReduction[3]* GVL_SetupMotorParameters.g_motorTrqConst[3] * 5000/1000;
END_METHOD

END_FUNCTION_BLOCK

// ---- FBs_Robots/FB_SetupArm.TcPOU
FUNCTION_BLOCK FB_SetupArm
VAR_INPUT
END_VAR
VAR_OUTPUT
END_VAR
VAR
	// arm index, from 1 to 4
	m_armIdx: INT;
	
	// joints
	m_joints :ARRAY[1..g_setupJntNum] OF FB_SetupJoint;
	
	// adjust detect
	m_adjustIO AT%I* :UDINT;
	m_manualAdjustOnFlag :BOOL;
	m_jnt5AdjustDir :INT; // -1, 0, 1;
	m_manualAdjustDetect : FB_setupAdjustDetect;
	m_jnt5AdjustDetect : FB_setupJnt5AdjustDetect;
	
	// arm cartesian data, defined in cart origin
	m_curCartPose	:ST_Frame;
	
	// cartesion position of remote center
	m_rcPos :Vec3d;	
	
	// arm joint data
	m_curMotorPos :Vec5d;
	m_curLinkPos :Vec5d;
	m_curJntPos :Vec5d;
	m_curJntVel :Vec5d;
	m_curJntTrq :Vec5d;
	m_rawJntCurrent :Vec5d;
	m_filtJntCurrent :Vec5d;
	m_cmdJntCurrent : Vec5d;
	m_cmdJntPos :Vec5d;
	m_cmdJntVel :Vec5d;
	m_cmdJntTrq :Vec5d;
		
	// arm gravity
	m_jntGravity : Vec5d:=g_zeroVec5d;
	
	// joint position controller
	m_jntPIDCtrl :ARRAY[1..g_setupJntNum] OF FB_PID;
	
	//arm light out to drive
	m_lightIO AT %Q* :DINT;
	
	// output arm light
	m_SdoWrite:ARRAY [1..2] OF FB_EcCoESdoWrite;
	
	//IP of operating arm
	m_armNetId:T_AmsNetId; 	
	
	//Joint port number
	m_jointAddrJ8:UINT;	
	m_jointAddrPbox:UINT;
	
END_VAR

PROPERTY armIdx : int
GET
armIdx:=m_armIdx;
END_GET
END_PROPERTY

METHOD PROTECTED checkIO : BOOL
VAR_INPUT
END_VAR
// check manual and auto adjust button
m_manualAdjustOnFlag := m_manualAdjustDetect.run(m_adjustIO);
m_jnt5AdjustDir := m_jnt5AdjustDetect.run(m_adjustIO);
END_METHOD

METHOD checkLight : BOOL
VAR_INPUT
	i_lightCtrlWord : UDINT;
END_VAR

VAR
	lightCtrlWord : UDINT;
END_VAR
// to PDO
m_lightIO := UDINT_TO_DINT(i_lightCtrlWord);

// trig sdo write
lightCtrlWord := SHL(i_lightCtrlWord,16);
m_SdoWrite[1](sNetId:= m_armNetId, nSlaveAddr:= m_jointAddrJ8, nSubIndex:= 0, nIndex:= 16#6085, pSrcBuf:=ADR(lightCtrlWord) , cbBufLen:=SIZEOF(lightCtrlWord) , bExecute:= TRUE, tTimeout:= , bBusy=> , bError=> , nErrId=> );
m_SdoWrite[2](sNetId:= m_armNetId, nSlaveAddr:= m_jointAddrPbox, nSubIndex:= 0, nIndex:= 16#6097, pSrcBuf:= ADR(lightCtrlWord), cbBufLen:= SIZEOF(lightCtrlWord), bExecute:= TRUE, tTimeout:= , bBusy=> , bError=> , nErrId=> );

// disable sdo write
IF NOT m_SdoWrite[1].bBusy AND  NOT m_SdoWrite[2].bBusy THEN
	m_SdoWrite[1](bExecute:=FALSE);
	m_SdoWrite[2](bExecute:=FALSE);
END_IF
END_METHOD

PROPERTY cmdJntCurrent : REFERENCE TO  Vec5d
GET
cmdJntCurrent ref= m_cmdJntCurrent;
END_GET
END_PROPERTY

PROPERTY curCartPose : REFERENCE TO ST_Frame
GET
curCartPose ref=m_curCartPose;
END_GET
END_PROPERTY

PROPERTY curJntPos : REFERENCE TO Vec5d
GET
curJntPos ref=m_curJntPos;
END_GET
END_PROPERTY

PROPERTY curJntTrq : REFERENCE TO Vec5d
GET
curJntTrq ref=m_curJntTrq;
END_GET
END_PROPERTY

PROPERTY curJntVel :REFERENCE TO Vec5d
GET
curJntVel ref=m_curJntVel;
END_GET
END_PROPERTY

PROPERTY curLinkPos :REFERENCE TO Vec5d
GET
curLinkPos ref=m_curLinkPos;
END_GET
END_PROPERTY

PROPERTY curMotorPos : REFERENCE TO  Vec5d
GET
curMotorPos ref=m_curMotorPos;
END_GET
END_PROPERTY

METHOD PUBLIC enable : BOOL
VAR_IN_OUT CONSTANT
	i_jntIdx :Vec5i;
END_VAR
VAR
	i :INT ;
END_VAR
FOR i:=1 TO g_setupJntNum DO
	IF 1= i_jntIdx[i] THEN
		m_joints[i].enable();
	ELSE
		m_joints[i].disable();
	END_IF
END_FOR
END_METHOD

PROPERTY filtJntCurrent :REFERENCE TO Vec5d
GET
filtJntCurrent ref= m_filtJntCurrent;
END_GET
END_PROPERTY

// compute cartesion pose in cart origin
METHOD PROTECTED forwardKinematic : BOOL
VAR_IN_OUT CONSTANT
	i_jntPos :Vec5d;
END_VAR
VAR_IN_OUT
	r_cartPose :ST_Frame;
	
	// position of remote center
	r_rcPos :Vec3d;
END_VAR
VAR
	a2,d4,d6:LREAL; //DH parameters
	
	Radius,Angle,R1,q:LREAL; //Disk structure parameters
	x,y,z:LREAL;
	basePosMatrix:ARRAY[1..4,1..4] OF LREAL;//transform from origin to C0
	
	T_50:ARRAY[1..4,1..4] OF LREAL; //transform from C0 to C5
	F5:ARRAY[1..4,1..4] OF LREAL; //transform from origin to C5
	q1,q2,q3,q4,q5:LREAL;	
	c14,s14,c5,s5,s1,c1:LREAL;
	
	fixPointTransform:ARRAY[1..4,1..4] OF LREAL; //transform from C5 to fixed point
	fixPointMatrix:ARRAY[1..4,1..4] OF LREAL;
END_VAR
//TODO: move DH parameter to GVL 


//****************input:five joint position of SetupArm********************//
q1:=i_jntPos[1]; q2:=i_jntPos[2]; q3:=i_jntPos[3]; q4:=i_jntPos[4]; q5:=i_jntPos[5];

//**********************DH parameters*************************//
IF (m_armIdx=1) THEN
	a2:=0.019; d4:=0.5205;
	
ELSIF (m_armIdx=2) THEN
	a2:=0.136; d4:=0.3545;
	
ELSIF (m_armIdx=3) THEN	
	a2:=0.136; d4:=0.3545;
	
ELSIF (m_armIdx=4) THEN	
	a2:=0.1825; d4:=0.5205;
END_IF
d6:=0.6387229+0.1659;

//********************transform form origin to C0***********************//
Radius:=0.170; Angle:=60.0*g_deg2Rad;
R1:=Radius;  q:=Angle;
IF (m_armIdx=1) THEN
	x:=-R1; y:=0; z:=0;
	
ELSIF (m_armIdx=2) THEN
	x:=-R1*COS(q); y:=-R1*SIN(q); z:=0;
	
ELSIF (m_armIdx=3) THEN	
	x:=R1*COS(q); y:=-R1*SIN(q); z:=0;
	
ELSIF (m_armIdx=4) THEN	
	x:=R1; y:=0; z:=0;
END_IF

basePosMatrix[1,1]:=0;
basePosMatrix[2,1]:=1;
basePosMatrix[3,1]:=0;
basePosMatrix[4,1]:=0;

basePosMatrix[1,2]:=-1;
basePosMatrix[2,2]:=0;
basePosMatrix[3,2]:=0;
basePosMatrix[4,2]:=0;

basePosMatrix[1,3]:=0;
basePosMatrix[2,3]:=0;
basePosMatrix[3,3]:=1;
basePosMatrix[4,3]:=0;

basePosMatrix[1,4]:=x;
basePosMatrix[2,4]:=y;
basePosMatrix[3,4]:=z;
basePosMatrix[4,4]:=1;

//***************output1:C5 posture relative to origin(other than C0)*************//
c14:=COS(q1+q4); s14:=SIN(q1+q4); 
c5:=COS(q5); s5:=SIN(q5);
c1:=COS(q1); s1:=SIN(q1);

T_50[1,1]:=c14*c5; 
T_50[2,1]:=s14*c5; 
T_50[3,1]:=-s5; 
T_50[4,1]:=0;

T_50[1,2]:=-c14*s5;
T_50[2,2]:=-s14*s5; 
T_50[3,2]:=-c5; 
T_50[4,2]:=0;

T_50[1,3]:=-s14;
T_50[2,3]:=c14;
T_50[3,3]:=0;
T_50[4,3]:=0;

T_50[1,4]:=a2*c1 + q2*s1;
T_50[2,4]:=a2*s1 - q2*c1;
T_50[3,4]:=d4 + q3;
T_50[4,4]:=1;

matMultiply(basePosMatrix,T_50,F5);
r_cartPose.m_pos[1]:=F5[1,4]; r_cartPose.m_pos[2]:=F5[2,4]; r_cartPose.m_pos[3]:=F5[3,4];

r_cartPose.m_rot[1,1]:=F5[1,1];  r_cartPose.m_rot[1,2]:=F5[1,2];  r_cartPose.m_rot[1,3]:=F5[1,3];
r_cartPose.m_rot[2,1]:=F5[2,1];  r_cartPose.m_rot[2,2]:=F5[2,2];  r_cartPose.m_rot[2,3]:=F5[2,3];
r_cartPose.m_rot[3,1]:=F5[3,1];  r_cartPose.m_rot[3,2]:=F5[3,2];  r_cartPose.m_rot[3,3]:=F5[3,3];

//********************output2:remote center position************************//
fixPointTransform[1,1]:=1;  fixPointTransform[2,2]:=1;  fixPointTransform[3,3]:=1;  fixPointTransform[4,4]:=1;  
fixPointTransform[2,4]:=-d6;  
matMultiply(F5,fixPointTransform,fixPointMatrix);
r_rcPos[1]:=fixPointMatrix[1,4];  r_rcPos[2]:=fixPointMatrix[2,4];  r_rcPos[3]:=fixPointMatrix[3,4];
END_METHOD

METHOD PUBLIC init : BOOL
VAR_INPUT
	i_armIdx:INT;
END_VAR
VAR 
	i :INT ;
	currentRatioMotor2Jnt:LREAL;
END_VAR
// arm statues init
m_armIdx:=i_armIdx;

// joint init
FOR i:=1 TO g_setupJntNum DO
	m_joints[i].init(m_armIdx, i,g_setupArmCtrlCycleTime);
END_FOR

// joint init
FOR i:=1 TO g_setupJntNum DO
	m_joints[i].initJntPos();
END_FOR

// update arm status if joint position is re-init
updateStatus();

// joint controller init
FOR i:=1 TO g_setupJntNum DO 
	currentRatioMotor2Jnt:=GVL_SetupMotorParameters.g_motorTrqConst[i]*GVL_SetupMotorParameters.g_motorReduction[i]/1000;
	m_jntPIDCtrl[i].init(g_setupArmCtrlCycleTime,GVL_SetupControlParameters.g_posKp[i],GVL_SetupControlParameters.g_posKd[i],
		GVL_SetupControlParameters.g_posKi[i], GVL_SetupControlParameters.g_posKiLimit[i]* currentRatioMotor2Jnt,
		GVL_SetupControlParameters.g_posCtrlLimit[i]*currentRatioMotor2Jnt);
END_FOR

//init arm netID and adrr
m_armNetId := GVL_SlaveJointEncoderCaliData.g_slaveArmNetID[armIdx];
m_jointAddrJ8 := GVL_SlaveJointEncoderCaliData.g_slaveJointNetPort[armIdx,3];
m_jointAddrPbox := GVL_SlaveJointEncoderCaliData.g_slaveJointNetPort[armIdx,4];
END_METHOD

METHOD PUBLIC isEnabled : BOOL
VAR_IN_OUT CONSTANT
	i_jntIdx :Vec5i;
END_VAR
VAR
	i :INT ;
END_VAR
isEnabled := TRUE;
FOR i:=1 TO g_setupJntNum DO
	IF 1= i_jntIdx[i] THEN
		isEnabled :=  (m_joints[i].isEnabled() AND isEnabled);
	END_IF
END_FOR
END_METHOD

PROPERTY jnt5AdjustDir : int
GET
jnt5AdjustDir := m_jnt5AdjustDir;
END_GET
END_PROPERTY

PROPERTY jntGravity :REFERENCE TO Vec5d
GET
jntGravity ref=m_jntGravity;
END_GET
END_PROPERTY

PROPERTY manualAdjustOn : bool
GET
manualAdjustOn := m_manualAdjustOnFlag;
END_GET
END_PROPERTY

PROPERTY rawJntCurrent :REFERENCE TO Vec5d
GET
rawJntCurrent ref=m_rawJntCurrent;
END_GET
END_PROPERTY

PROPERTY rcPos :REFERENCE to Vec3d
GET
rcPos REF= m_rcPos;
END_GET
END_PROPERTY

// update joints control command
METHOD PUBLIC updateCmds : BOOL
VAR_IN_OUT CONSTANT
	i_armCtrlCmd : ST_SetupArmCtrlCmds;
END_VAR
VAR
	i:INT;
END_VAR
m_cmdJntTrq:=i_armCtrlCmd.m_cmdJntTrq;
m_cmdJntPos :=i_armCtrlCmd.m_cmdJntPos;
m_cmdJntVel :=i_armCtrlCmd.m_cmdJntVel;

// enable/disable joints
enable(i_armCtrlCmd.m_jntEnableFlag);

// position/torque control
FOR i:=1 TO g_setupJntNum DO 
	IF i_armCtrlCmd.m_jntOPMode[i]=DriverOPMode_PosTrq THEN
		// position controller and gravity feedforward
		m_cmdJntTrq[i]:=m_jntPIDCtrl[i].run(m_cmdJntPos[i],m_curJntPos[i],0,m_curJntVel[i]);
		m_cmdJntTrq[i]:=m_cmdJntTrq[i]+m_jntGravity[i];
		m_joints[i].updateCmds(DriverOPMode_Trq,m_cmdJntPos[i],m_cmdJntTrq[i]);
	ELSIF i_armCtrlCmd.m_jntOPMode[i]=DriverOPMode_Trq THEN
		// gravity feedforward
		m_jntPIDCtrl[i].reset();
		m_cmdJntTrq[i]:=m_cmdJntTrq[i]+m_jntGravity[i]+GVL_SetupArmDynamics.g_setupJntGravityOffset[m_armIdx, i];
		m_joints[i].updateCmds(DriverOPMode_Trq,i_armCtrlCmd.m_cmdJntPos[i],m_cmdJntTrq[i]);
	ELSE
		m_jntPIDCtrl[i].reset();
		m_cmdJntTrq[i]:=0;
		m_joints[i].updateCmds(DriverOPMode_Pos,i_armCtrlCmd.m_cmdJntPos[i],m_cmdJntTrq[i]);
	END_IF
	
END_FOR
END_METHOD

METHOD PUBLIC updateDyna : BOOL
VAR_IN_out constant
	i_jnt3Gravity :LREAL;
	i_jnt5Gravity :LREAL;
END_VAR
m_jntGravity[3]:=i_jnt3Gravity;
m_jntGravity[5]:=i_jnt5Gravity;
END_METHOD

// update arm status, including kinematic and dynamic
METHOD PUBLIC updateStatus : BOOL
VAR_INPUT
END_VAR
VAR 
	i,j:INT;
END_VAR
// update joint data
FOR i:=1 TO g_setupJntNum DO
	m_joints[i].updateStatus();
END_FOR

// check adjust button
checkIO();

// get joint data
FOR i:=1 TO g_setupJntNum DO
	m_curMotorPos[i]:=m_joints[i].motorPos;
	m_curLinkPos[i]:=m_joints[i].linkPos;
	m_curJntPos[i]:=m_joints[i].jntPos;
	m_curJntVel[i]:=m_joints[i].jntVel;
	m_curJntTrq[i]:=m_joints[i].jntTrq;
	m_rawJntCurrent[i]:=m_joints[i].rawCurrent;
	m_filtJntCurrent[i]:=m_joints[i].filtCurrent;
	m_cmdJntCurrent[i]:=m_joints[i].cmdCurrent;
END_FOR 

// cartesion pose
forwardKinematic(m_curJntPos,m_curCartPose,m_rcPos);
END_METHOD

END_FUNCTION_BLOCK

// ---- FBs_Robots/FB_SlaveJoint.TcPOU
FUNCTION_BLOCK FB_SlaveJoint EXTENDS FB_JointBase
VAR_INPUT
END_VAR
VAR_OUTPUT
END_VAR
VAR
	// power box joint motor rated current
	m_wristJntRatedCurrent : DINT := 200;

END_VAR

METHOD PUBLIC init : BOOL
VAR_INPUT
	i_armIdx :INT;
	i_jntIdx :INT;
	i_controlCycleTime :LREAL;
	// velocity is calculated every (m_velCalcCycles) control cycles
	// TODO: insturment joint motor can not reach 4k now, so calculate their velocity with 1k frequency, need to remove later
	i_velCalcCycles :INT;
END_VAR
m_armIdx:=i_armIdx;
m_jntIdx:=i_jntIdx;
m_cycleTime := i_controlCycleTime;
m_velCalcCycles :=MAX(i_velCalcCycles,1);

IF m_armIdx =3 THEN
	m_linkEncoderRes :=GVL_SlaveMotorParameters.g_absEncoderResFR[i_jntIdx];
	m_linkEncoderDir :=GVL_SlaveJointEncoderCaliData.g_asbEncoderDirFR[i_jntIdx];
	m_linkEncLimitBuffer := GVL_SlaveJointEncoderCaliData.g_linkEncLimitBufferFR[i_jntIdx];
ELSE
	m_linkEncoderRes :=GVL_SlaveMotorParameters.g_absEncoderRes[i_jntIdx];
	m_linkEncoderDir :=GVL_SlaveJointEncoderCaliData.g_asbEncoderDir[i_jntIdx];
	m_linkEncLimitBuffer := GVL_SlaveJointEncoderCaliData.g_linkEncLimitBuffer[i_jntIdx];
END_IF

// hardware parameters
m_motorEncoderRes :=GVL_SlaveMotorParameters.g_incEncoderRes[i_jntIdx];
//m_linkEncoderRes :=GVL_SlaveMotorParameters.g_absEncoderRes[i_jntIdx];
m_motorReduction :=GVL_SlaveMotorParameters.g_motorReduction[i_jntIdx];
m_linkEncoderReduction :=GVL_SlaveMotorParameters.g_absEncoderReduction[i_jntIdx];
m_trqConst :=GVL_SlaveMotorParameters.g_motorTrqConst[i_jntIdx];
m_maxCurrent :=GVL_SlaveMotorParameters.g_motorMaxCurrent[i_jntIdx];
m_motorDir :=GVL_SlaveMotorParameters.g_motorDir[i_jntIdx];								
m_minJntPos	:=GVL_SlaveMotorParameters.g_minJntPos[i_jntIdx];
m_maxJntPos	:=GVL_SlaveMotorParameters.g_maxJntPos[i_jntIdx];

//link encoder calibartion data
//m_linkEncoderDir :=GVL_SlaveJointEncoderCaliData.g_asbEncoderDir[i_jntIdx];
m_minLinkEncoder :=GVL_SlaveJointEncoderCaliData.g_minLinkEncoder[i_armIdx, i_jntIdx] - m_linkEncoderDir*m_linkEncLimitBuffer; // expand limit
m_maxLinkEncoder :=GVL_SlaveJointEncoderCaliData.g_maxLinkEncoder[i_armIdx, i_jntIdx] + m_linkEncoderDir*m_linkEncLimitBuffer; // expand limit
m_caliLinkEncoder :=GVL_SlaveJointEncoderCaliData.g_caliLinkEncoder[i_armIdx, i_jntIdx];
m_linkEncCaliJntPos :=GVL_SlaveJointEncoderCaliData.g_linkEncCaliJntPos[i_jntIdx];
m_linkEncZeroCross :=GVL_SlaveJointEncoderCaliData.g_linkEncZeroCross[i_armIdx, i_jntIdx];
m_multiCycles :=GVL_SlaveJointEncoderCaliData.g_multipleCyclesJoint[i_armIdx,i_jntIdx];

// convert cali link encoder if joint cross zero
IF 1=m_linkEncZeroCross THEN
	IF 1=m_linkEncoderDir AND m_caliLinkEncoder < m_minLinkEncoder THEN
		m_caliLinkEncoder := GVL_SlaveJointEncoderCaliData.g_caliLinkEncoder[i_armIdx, i_jntIdx] + m_linkEncoderRes;
	ELSIF -1=m_linkEncoderDir AND m_caliLinkEncoder < m_maxLinkEncoder THEN
		m_caliLinkEncoder := GVL_SlaveJointEncoderCaliData.g_caliLinkEncoder[i_armIdx, i_jntIdx] + m_linkEncoderRes;
	END_IF
END_IF

// macro data
m_trq2CurrentRatio:=m_motorDir * 1000.0/(m_trqConst*m_motorReduction);
m_current2TrqRatio:=m_motorDir * (m_trqConst*m_motorReduction)/1000.0;
m_linkEnc2PosRatio := 2*PI*m_linkEncoderDir/(m_linkEncoderReduction*m_linkEncoderRes);
m_motorEnc2PosRatio := 2*PI * m_motorDir/(m_motorReduction * m_motorEncoderRes);

// motor data init
m_rawJntVel :=0;
m_curJntVel:=0;
m_curJntTrq :=0;
m_rawCurrent :=0;
m_filtCurrent :=0;
m_cmdJntVel :=0.0;
m_cmdJntTrq :=0.0;
m_cmdCurrent := 0.0;

// filter init
m_jntVelLpf.init(1, GVL_SlaveControlParameters.g_curJntVelLpfCutoffFreq, g_slaveArmCtrlFreq/m_velCalcCycles);
m_cmdTrqLpf.init(1, GVL_SlaveControlParameters.g_cmdJntTrqLpfCutoffFreq, g_slaveArmCtrlFreq);
m_curTrqLpf.init(1, GVL_SlaveControlParameters.g_curJntTrqLpfCutoffFreq, g_slaveArmCtrlFreq);

// driver init value
m_motorOutputs.m_controlWord:=DriverCtrlWord_INIT;
m_motorOutputs.m_opMode:=INT_TO_SINT(DriverOPMode_Pos);
m_motorOutputs.m_cmdCurrent:=0;
m_motorOutputs.m_cmdMotorEncoder:=m_motorInputs.m_motorEncoder;
END_METHOD

METHOD PUBLIC updateCmds : BOOL
VAR_INPUT
	i_opMode : E_DriverOPMode;
	i_cmdPos :LREAL;
	i_cmdTrq :LREAL;
END_VAR
VAR
	filtCmdTrq :LREAL;
END_VAR
SUPER^.updateCmds(i_opMode, i_cmdPos, i_cmdTrq);

// write SDO data
//writeSDOData();
END_METHOD

METHOD PROTECTED writeSDOData : BOOL
VAR_INPUT
END_VAR
VAR
	SDOSubIndexMode :WORD;
	SDOSubIndexCur :WORD;
END_VAR
//动力盒移动关节和器械旋转关节，共享一个控制字，由SDO写入
IF (m_jntIdx=3) OR (m_jntIdx=8)  THEN
	SDOSubIndexMode :=16#609B;
	SDOSubIndexCur:=16#6098;
//动力盒3、5号电机为一个驱动器，共享一个控制字，由SDO写入
ELSIF (m_jntIdx=4) OR (m_jntIdx=6)  THEN
	SDOSubIndexMode :=16#609C;
	SDOSubIndexCur:=16#6099;
//动力盒2、4号电机为一个驱动器，共享一个控制字，由SDO写入
ELSIF (m_jntIdx=5) OR (m_jntIdx=7)  THEN
	SDOSubIndexMode :=16#609D;
	SDOSubIndexCur:=16#609A;
END_IF

IF m_jntIdx <3 THEN
	RETURN;
END_IF

// write driver operation mode if it changs
IF  m_jntIdx >=3 AND m_jntIdx <=8 THEN
	m_opModeSDOWrite(sNetID:= GVL_SlaveJointEncoderCaliData.g_slaveArmNetID[m_armIdx],
					nSlaveAddr := GVL_SlaveJointEncoderCaliData.g_slaveJointNetPort[m_armIdx,m_jntIdx],
					nSubIndex:=0,nIndex:=SDOSubIndexMode,pSrcBuf:=ADR(m_motorOutputs.m_opMode),cbBufLen:=SIZEOF(m_motorOutputs.m_opMode),bExecute:=TRUE);
	IF NOT m_opModeSDOWrite.bBusy THEN
		m_opModeSDOWrite(bExecute:=FALSE);
	END_IF
END_IF

// write max motor current if it changes and works in position mode
IF m_jntIdx >=4 AND m_jntIdx <=8  THEN 
	m_MotorCurrentSDOWrite(sNetID:= GVL_SlaveJointEncoderCaliData.g_slaveArmNetID[m_armIdx],
					nSlaveAddr := GVL_SlaveJointEncoderCaliData.g_slaveJointNetPort[m_armIdx,m_jntIdx],
					nSubIndex:=0,nIndex:=SDOSubIndexCur,pSrcBuf:=ADR(m_wristJntRatedCurrent),cbBufLen:=SIZEOF(m_wristJntRatedCurrent),bExecute:=TRUE);
	IF NOT m_MotorCurrentSDOWrite.bBusy THEN
		m_MotorCurrentSDOWrite(bExecute:=FALSE);
	END_IF
END_IF
END_METHOD

END_FUNCTION_BLOCK

// ---- FBs_SetupControllers/FB_SetupCtrlManualAdjust.TcPOU
// Brief: Setup Arm Adjust
FUNCTION_BLOCK PUBLIC FB_SetupCtrlManualAdjust EXTENDS FB_SetupArmCtrlBase
VAR_INPUT
END_VAR
VAR_OUTPUT
END_VAR
VAR
	// friction compensation scale
	m_frictionScale :LREAL :=0.5;
	
	// velocity threshold for friction compensation 
	m_jnt3FrictionCompVelLow :LREAL := 0.0005;
	m_frictionScaleLow :LREAL :=0.3;
	m_jnt3FrictionCompVelMiddle :LREAL := 0.005;
	m_frictionScaleMiddle :LREAL :=0.5;
	m_jnt3FrictionCompVelHigh :LREAL := 0.05;
	m_frictionScaleHigh :LREAL :=0.7;
	
	// jnt5 adjust velocity
	m_jnt5MaxAdjustVel :LREAL:=5.0*g_deg2Rad;
	m_jnt5MaxAdjustAcc :LREAL:=60*g_deg2Rad;
	
	// jnt5 enabled time period
	m_jnt5EnableTime :LREAL :=0;
	
	// time threshold to drive jnt5 after it's enabled
	m_jnt5AdjustWaitTime :LREAL := 0.25;

	// distance buffer from joint limit to start damp
	m_limitBufferForDamp :LREAL :=0.05;
	
	// max damp
	m_maxDamp :LREAL := 3000;
	
	m_limitBufferForCtrl : LREAL := 0.01;
END_VAR

// override this function in each exact controller
METHOD PROTECTED calcCmdJntPos : BOOL
VAR_IN_OUT CONSTANT
	i_setupArm	:FB_SetupArm;
END_VAR


VAR 
	i :INT;
END_VAR
// enable/disenable joint5
IF i_setupArm.jnt5AdjustDir = 0 THEN
	m_jntEnableFlag[5] := 0;
	m_cmdJntPos[5]:=i_setupArm.curJntPos[5];
	m_jnt5EnableTime:=0;
	m_cmdJntVel[5]:=0;
	RETURN;
ELSE
	// disable joints if this joint is an unrecoverable failure
	m_jntEnableFlag[5] :=  BOOL_TO_INT( NOT (SafetyCheck.m_SafetyCheck.m_jntErrFlag[i_setupArm.armIdx, 0, 3] OR  SafetyCheck.m_SafetyCheck.m_jntErrFlag[i_setupArm.armIdx, 5, 3]));
	m_jnt5EnableTime := m_jnt5EnableTime + g_setupArmCtrlCycleTime;
END_IF

// update command position
IF m_jnt5EnableTime>m_jnt5AdjustWaitTime THEN
	m_cmdJntVel[5]:=m_cmdJntVel[5] + i_setupArm.jnt5AdjustDir * m_jnt5MaxAdjustAcc * g_setupArmCtrlCycleTime;
	m_cmdJntVel[5]:=LIMIT(-m_jnt5MaxAdjustVel, m_cmdJntVel[5], m_jnt5MaxAdjustVel);
	
	// joint limit
	IF (m_cmdJntPos[5] > GVL_SetupMotorParameters.g_maxJntPos[i_setupArm.armIdx, 5] - g_setupJntPosLimitBuffer[5] AND m_cmdJntVel[5]>0) OR 
		(m_cmdJntPos[5] < GVL_SetupMotorParameters.g_minJntPos[i_setupArm.armIdx, 5] + g_setupJntPosLimitBuffer[5] AND m_cmdJntVel[5]<0)  THEN
		m_cmdJntVel[5] := 0;
	END_IF
	
	m_cmdJntPos[5]:= m_cmdJntPos[5] + m_cmdJntVel[5] * g_setupArmCtrlCycleTime;
END_IF
END_METHOD

// override this function in each exact controller
METHOD PROTECTED calcCmdJntTrq : BOOL
VAR_IN_OUT CONSTANT
	i_setupArm	:FB_SetupArm;
END_VAR
VAR
	i:INT;
	vel :LREAL;
	scale:LREAL;
	ratio:LREAL;
	dampScale :LREAL;
	limitDis:LREAL;
	dampOffset : LREAL;
END_VAR
// set joint torque to zero in default
m_cmdJntTrq := g_zeroVec5d;

//enable/diable  joint1-4
IF NOT(i_setupArm.manualAdjustOn) THEN
	FOR i:=1 TO 4 DO
		m_jntEnableFlag[i] := 0;
		m_jntOPMode[i]:=DriverOPMode_Pos;
	END_FOR
	
	// TODO: setup joint3 would "jump" a bit when transit from torque mode to position mode
	m_jntOPMode[3] := DriverOPMode_Trq;
	RETURN;
ELSE
	FOR i:=1 TO 4 DO
		// disable joints if this joint is an unrecoverable failure
		m_jntEnableFlag[i] := BOOL_TO_INT( NOT (SafetyCheck.m_SafetyCheck.m_jntErrFlag[i_setupArm.armIdx, 0, 3] OR  SafetyCheck.m_SafetyCheck.m_jntErrFlag[i_setupArm.armIdx, i, 3]));
		m_jntOPMode[i]:=DriverOPMode_Trq;
		m_cmdJntPos[i] := i_setupArm.curJntPos[i];
	END_FOR
END_IF

// friction scale
vel:=ABS(i_setupArm.curJntVel[3]);
IF vel < m_jnt3FrictionCompVelLow THEN
	m_frictionScale := m_frictionScaleLow * vel/m_jnt3FrictionCompVelLow ;
ELSIF  vel > m_jnt3FrictionCompVelLow AND vel  < m_jnt3FrictionCompVelMiddle THEN
	ratio:= (vel-m_jnt3FrictionCompVelLow)/(m_jnt3FrictionCompVelMiddle-m_jnt3FrictionCompVelLow);
	m_frictionScale :=m_frictionScaleLow+ratio * (m_frictionScaleMiddle-m_frictionScaleLow);
ELSIF  vel > m_jnt3FrictionCompVelMiddle AND vel  < m_jnt3FrictionCompVelHigh THEN
	ratio:= (vel-m_jnt3FrictionCompVelMiddle)/(m_jnt3FrictionCompVelHigh-m_jnt3FrictionCompVelMiddle);
	m_frictionScale :=m_frictionScaleMiddle+ratio * (m_frictionScaleHigh-m_frictionScaleMiddle);
ELSIF  vel > m_jnt3FrictionCompVelHigh THEN
	m_frictionScale := m_frictionScaleHigh;
END_IF

// add damp near joint limit 
IF (i_setupArm.curJntPos[3] > GVL_SetupMotorParameters.g_maxJntPos[1,3] - m_limitBufferForCtrl ) 
	OR (i_setupArm.curJntPos[3] < GVL_SetupMotorParameters.g_minJntPos[1,3] + m_limitBufferForCtrl) OR CartControl.m_cartRobot.m_slaveCart.m_columnAdjustEnable  THEN
	dampOffset:= 0;
ELSIF (i_setupArm.curJntPos[3] > GVL_SetupMotorParameters.g_maxJntPos[1,3] - m_limitBufferForDamp AND  i_setupArm.curJntVel[3]> 0 ) 
	OR (i_setupArm.curJntPos[3] < GVL_SetupMotorParameters.g_minJntPos[1,3] + m_limitBufferForDamp AND  i_setupArm.curJntVel[3]<0 )  THEN
	limitDis := MIN(GVL_SetupMotorParameters.g_maxJntPos[1,3] - i_setupArm.curJntPos[3], i_setupArm.curJntPos[3]-GVL_SetupMotorParameters.g_minJntPos[1,3]);
	dampScale  :=LIMIT(0, 1-limitDis/(m_limitBufferForDamp-m_limitBufferForCtrl),1);
	dampOffset:= -dampScale * m_maxDamp * i_setupArm.curJntVel[3];
END_IF


// add friction compensation
m_frictionScale := LIMIT(0, m_frictionScale, 1);
m_cmdJntTrq[3]:= 0;// m_frictionScale * sign(i_setupArm.curJntVel[3])*jnt3Friction(i_setupArm.armIdx, i_setupArm.curJntPos[3]) + dampOffset;
END_METHOD

METHOD PUBLIC init : BOOL
VAR_IN_OUT CONSTANT
	i_setupArm	:FB_SetupArm;
END_VAR
VAR_IN_OUT 
	r_setupArmCtrlCmd :ST_SetupArmCtrlCmds;
END_VAR
SUPER^.Init(i_setupArm,r_setupArmCtrlCmd);
m_jnt5EnableTime :=0;
END_METHOD

METHOD PROTECTED jnt3Friction : Lreal
VAR_INPUT
	i_armIdx:INT;
	i_jnt3Pos :LREAL;
END_VAR

VAR
	q:LREAL;
END_VAR
q := LIMIT(GVL_SetupArmDynamics.g_setupJnt3GravityPosRange[i_armIdx,1], i_jnt3Pos, GVL_SetupArmDynamics.g_setupJnt3GravityPosRange[i_armIdx,2]);
jnt3Friction:=GVL_SetupArmDynamics.g_setupJnt3FrictionParams[i_armIdx,1]*EXPT(q,3)+GVL_SetupArmDynamics.g_setupJnt3FrictionParams[i_armIdx,2]*EXPT(q,2)+
				GVL_SetupArmDynamics.g_setupJnt3FrictionParams[i_armIdx,3]*q+GVL_SetupArmDynamics.g_setupJnt3FrictionParams[i_armIdx,4];
END_METHOD

END_FUNCTION_BLOCK
